               IF NOT "Valves_DB".Valve[#i].Healthy OR "Valves_DB".PositionFault[#i]
                  OR "Valves_DB".TimeoutOpenAlarm[#i] OR "Valves_DB".TimeoutCloseAlarm[#i]
                  OR "Valves_DB".UnexpMove[#i] OR "Valves_DB".PosLostTmr[#i].Q
                  OR "Valves_DB".DirFault[#i] THEN
                   "Valves_DB".StateCode[#i] := 1;
                   #tempFault := #tempFault + 1;
                   IF #i <= 27 THEN #tempAftFault := #tempAftFault + 1;
                   ELSIF #i <= 54 THEN #tempErFault := #tempErFault + 1;
                   ELSE #tempFwdFault := #tempFwdFault + 1;
                   END_IF;
               ELSIF "Valves_DB".Valve[#i].LocalMode THEN
                   "Valves_DB".StateCode[#i] := 2;
                   #tempLocal := #tempLocal + 1;
                   IF #i <= 27 THEN #tempAftLocal := #tempAftLocal + 1;
                   ELSIF #i <= 54 THEN #tempErLocal := #tempErLocal + 1;
                   ELSE #tempFwdLocal := #tempFwdLocal + 1;
                   END_IF;
               ELSIF "Valves_DB".Valve[#i].OpenValve THEN
                   // 6 = OPENING. The run latches are checked BEFORE the limit switches on purpose:
                   // what the system is doing to the valve outranks where the valve currently sits.
                   // Without this, a valve commanded CLOSE while still on its open limit displayed a
                   // settled green "FULLY OPEN" - no acknowledgement that the command had even
                   // registered on a normal stroke, and on a fault a confidently wrong indication for
                   // the full travel timeout. StateCode used to answer only "where is the valve";
                   // it now also answers "what is being done to it", which is the half that matters
                   // when something is going wrong.
                   "Valves_DB".StateCode[#i] := 6;
                   #tempTransit := #tempTransit + 1;
                   IF #i <= 27 THEN #tempAftTransit := #tempAftTransit + 1;
                   ELSIF #i <= 54 THEN #tempErTransit := #tempErTransit + 1;
                   ELSE #tempFwdTransit := #tempFwdTransit + 1;
                   END_IF;
               ELSIF "Valves_DB".Valve[#i].CloseValve THEN
                   "Valves_DB".StateCode[#i] := 7;   // 7 = CLOSING
                   #tempTransit := #tempTransit + 1;
                   IF #i <= 27 THEN #tempAftTransit := #tempAftTransit + 1;
                   ELSIF #i <= 54 THEN #tempErTransit := #tempErTransit + 1;
                   ELSE #tempFwdTransit := #tempFwdTransit + 1;
                   END_IF;
               ELSIF "Valves_DB".Valve[#i].OpenFB AND NOT "Valves_DB".Valve[#i].ClosedFB THEN
                   "Valves_DB".StateCode[#i] := 3;
                   #tempOpen := #tempOpen + 1;
                   IF #i <= 27 THEN #tempAftOpen := #tempAftOpen + 1;
                   ELSIF #i <= 54 THEN #tempErOpen := #tempErOpen + 1;
                   ELSE #tempFwdOpen := #tempFwdOpen + 1;
                   END_IF;
               ELSIF NOT "Valves_DB".Valve[#i].OpenFB AND "Valves_DB".Valve[#i].ClosedFB THEN
                   "Valves_DB".StateCode[#i] := 4;
                   #tempClosed := #tempClosed + 1;
                   IF #i <= 27 THEN #tempAftClosed := #tempAftClosed + 1;
                   ELSIF #i <= 54 THEN #tempErClosed := #tempErClosed + 1;
                   ELSE #tempFwdClosed := #tempFwdClosed + 1;
                   END_IF;
               ELSE
                   "Valves_DB".StateCode[#i] := 5;
                   #tempTransit := #tempTransit + 1; // MOVING state!
                   IF #i <= 27 THEN #tempAftTransit := #tempAftTransit + 1;
                   ELSIF #i <= 54 THEN #tempErTransit := #tempErTransit + 1;
                   ELSE #tempFwdTransit := #tempFwdTransit + 1;
                   END_IF;
               END_IF;
           ELSE
               "Valves_DB".StateCode[#i] := 0;
               "Valves_DB".PosCode[#i] := 0;
               "Valves_DB".DispCode[#i] := 0;
               "Valves_DB".FaultCode[#i] := 0;
               "Valves_DB".Valve[#i].OpenCmd := FALSE;
               "Valves_DB".Valve[#i].CloseCmd := FALSE;
               // Drop the run latches too. Without this, de-configuring a valve mid-travel (the popup's
               // SERVICE toggle reaches this from the HMI) left OpenValve/CloseValve latched TRUE with
               // no logic left managing them - and since FC_IoMapper skipped unconfigured valves, the
               // DQ bit kept its last value and FC_PhysicalIoCopy went on copying it to the real %Q
               // forever. The relay would have stayed energised indefinitely while the screen showed a
               // harmless-looking UNCONFIGURED. Paired with the FC_IoMapper change that now drives DQ
               // unconditionally, so clearing these actually de-energises the output.
               "Valves_DB".Valve[#i].OpenValve := FALSE;
               "Valves_DB".Valve[#i].CloseValve := FALSE;
               "Valves_DB".CmdPos[#i] := 0;
               // Don't let an unconfigured/removed valve leave a stale latched alarm behind.
               "Valves_DB".TimeoutOpenAlarm[#i] := FALSE;
               "Valves_DB".TimeoutCloseAlarm[#i] := FALSE;
               "Valves_DB".UnexpMove[#i] := FALSE;
               "Valves_DB".DirFault[#i] := FALSE;
               "Valves_DB".PrevOpenFB[#i] := FALSE;
               "Valves_DB".PrevClosedFB[#i] := FALSE;
           END_IF;
       END_FOR;

       "Valves_DB".TotalOpen := #tempOpen;
       "Valves_DB".TotalClosed := #tempClosed;
       "Valves_DB".TotalTransit := #tempTransit;
       "Valves_DB".TotalFault := #tempFault;
       "Valves_DB".TotalLocal := #tempLocal;
       "Valves_DB".TotalConfigured := #tempConfigured;

       "Valves_DB".ErOpen := #tempErOpen;
       "Valves_DB".ErClosed := #tempErClosed;
       "Valves_DB".ErTransit := #tempErTransit;
       "Valves_DB".ErFault := #tempErFault;
       "Valves_DB".ErLocal := #tempErLocal;
       "Valves_DB".ErConfigured := #tempErConfigured;

       "Valves_DB".FwdOpen := #tempFwdOpen;
       "Valves_DB".FwdClosed := #tempFwdClosed;
       "Valves_DB".FwdTransit := #tempFwdTransit;
       "Valves_DB".FwdFault := #tempFwdFault;
       "Valves_DB".FwdLocal := #tempFwdLocal;
       "Valves_DB".FwdConfigured := #tempFwdConfigured;

       "Valves_DB".AftOpen := #tempAftOpen;
       "Valves_DB".AftClosed := #tempAftClosed;
       "Valves_DB".AftTransit := #tempAftTransit;
       "Valves_DB".AftFault := #tempAftFault;
       "Valves_DB".AftLocal := #tempAftLocal;
       "Valves_DB".AftConfigured := #tempAftConfigured;

       // ---- Alarm condition bit-packing -----------------------------------------
       // WinCC discrete alarms trigger off a bit within a Word tag (RaisedStateTag +
       // RaisedStateTagBitNumber), not a bare Bool array element, so each of the 7 per-valve
       // conditions gets packed into 6 words (96 bits available, 89 used) here. Valve V's bit for any
       // condition is word (V-1)/16, bit (V-1) MOD 16 — matches how the HMI-side alarm creation
       // computes the same trigger address, so the two have to stay in lockstep.
       FOR #w := 0 TO 5 DO
           #packWord := 0;
           FOR #b := 0 TO 15 DO
               #bitIdx := #w * 16 + #b + 1;
               IF #bitIdx <= 89 THEN
                   IF "Valves_DB".Valve[#bitIdx].Configured AND NOT "Valves_DB".Valve[#bitIdx].Healthy THEN
                       #packWord := #packWord OR SHL(IN := W#16#1, N := INT_TO_UDINT(#b));
                   END_IF;
               END_IF;
           END_FOR;
           "Valves_DB".W_Unhealthy[#w] := #packWord;
       END_FOR;

       FOR #w := 0 TO 5 DO
           #packWord := 0;
           FOR #b := 0 TO 15 DO
               #bitIdx := #w * 16 + #b + 1;
               IF #bitIdx <= 89 THEN
                   IF "Valves_DB".Valve[#bitIdx].Configured AND "Valves_DB".Valve[#bitIdx].OpenFB AND "Valves_DB".Valve[#bitIdx].ClosedFB THEN
                       #packWord := #packWord OR SHL(IN := W#16#1, N := INT_TO_UDINT(#b));
                   END_IF;
               END_IF;
           END_FOR;
           "Valves_DB".W_Conflict[#w] := #packWord;
       END_FOR;

       FOR #w := 0 TO 5 DO
           #packWord := 0;
           FOR #b := 0 TO 15 DO
               #bitIdx := #w * 16 + #b + 1;
               IF #bitIdx <= 89 THEN
                   IF "Valves_DB".Valve[#bitIdx].Configured AND "Valves_DB".TimeoutOpenAlarm[#bitIdx] THEN
                       #packWord := #packWord OR SHL(IN := W#16#1, N := INT_TO_UDINT(#b));
                   END_IF;
               END_IF;
           END_FOR;
           "Valves_DB".W_FailOpen[#w] := #packWord;
       END_FOR;

       FOR #w := 0 TO 5 DO
           #packWord := 0;
           FOR #b := 0 TO 15 DO
               #bitIdx := #w * 16 + #b + 1;
               IF #bitIdx <= 89 THEN
                   IF "Valves_DB".Valve[#bitIdx].Configured AND "Valves_DB".TimeoutCloseAlarm[#bitIdx] THEN
                       #packWord := #packWord OR SHL(IN := W#16#1, N := INT_TO_UDINT(#b));
                   END_IF;
               END_IF;
           END_FOR;
           "Valves_DB".W_FailClose[#w] := #packWord;
       END_FOR;

       FOR #w := 0 TO 5 DO
           #packWord := 0;
           FOR #b := 0 TO 15 DO
               #bitIdx := #w * 16 + #b + 1;
               IF #bitIdx <= 89 THEN
                   IF "Valves_DB".Valve[#bitIdx].Configured AND "Valves_DB".PosLostTmr[#bitIdx].Q THEN
                       #packWord := #packWord OR SHL(IN := W#16#1, N := INT_TO_UDINT(#b));
                   END_IF;
               END_IF;
           END_FOR;
           "Valves_DB".W_LossPos[#w] := #packWord;
       END_FOR;

       FOR #w := 0 TO 5 DO
           #packWord := 0;
           FOR #b := 0 TO 15 DO
               #bitIdx := #w * 16 + #b + 1;
               IF #bitIdx <= 89 THEN
                   IF "Valves_DB".Valve[#bitIdx].Configured AND "Valves_DB".UnexpMove[#bitIdx] THEN
                       #packWord := #packWord OR SHL(IN := W#16#1, N := INT_TO_UDINT(#b));
                   END_IF;
               END_IF;
           END_FOR;
           "Valves_DB".W_UnexpMove[#w] := #packWord;
       END_FOR;

       FOR #w := 0 TO 5 DO
           #packWord := 0;
           FOR #b := 0 TO 15 DO
               #bitIdx := #w * 16 + #b + 1;
               IF #bitIdx <= 89 THEN
                   IF "Valves_DB".Valve[#bitIdx].Configured AND "Valves_DB".Valve[#bitIdx].LocalMode THEN
                       #packWord := #packWord OR SHL(IN := W#16#1, N := INT_TO_UDINT(#b));
                   END_IF;
               END_IF;
           END_FOR;
           "Valves_DB".W_Local[#w] := #packWord;
       END_FOR;

       // H: direction / limit-switch discrepancy.
       FOR #w := 0 TO 5 DO
           #packWord := 0;
           FOR #b := 0 TO 15 DO
               #bitIdx := #w * 16 + #b + 1;
               IF #bitIdx <= 89 THEN
                   IF "Valves_DB".Valve[#bitIdx].Configured AND "Valves_DB".DirFault[#bitIdx] THEN
                       #packWord := #packWord OR SHL(IN := W#16#1, N := INT_TO_UDINT(#b));
                   END_IF;
               END_IF;
           END_FOR;
           "Valves_DB".W_DirFault[#w] := #packWord;
       END_FOR;

       // Simulated hardware health (indices 1..9) into a single word.
       #packWord := 0;
       FOR #b := 0 TO 8 DO
           IF NOT "Valves_DB".HwHealthy[#b + 1] THEN
               #packWord := #packWord OR SHL(IN := W#16#1, N := INT_TO_UDINT(#b));
           END_IF;
       END_FOR;
       "Valves_DB".HwWord := #packWord;

       // ---- Paged table windows ------------------------------------------------
       // The HMI valve table has 14 fixed slots. Copy whichever page each zone is showing into
       // these windows so every HMI slot can bind to a constant tag name (e.g. ErTblState[3])
       // rather than building the name in JavaScript from a page tag — that indirection is what
       // forced the table onto ~126 polled scripts and made the screen slow to load.
       // TblState = -1 marks a slot with no valve on this page (0 already means UNCONFIGURED).
       // 14 iterations x 3 zones per scan is negligible next to the 89-valve loop above.

       // ── PAGED TABLE WINDOWS — gated, not rebuilt every scan ────────────────────────────
       // These four loops copy ~350 STRINGS per scan (tag, name, location, function, CmNo, VTag,
       // state text x 58 slots). String copies are the slowest thing in this program and were the
       // single biggest contributor to scan time, all to produce data no operator can read faster
       // than a few times a second.
       // So: rebuild on a 200 ms tick, OR immediately when a page changes. The page test matters -
       // waiting up to 200 ms after a page button would feel laggy, and paging is the one moment the
       // window contents change wholesale.
       #doWindows := #winTick
           OR ("Valves_DB".AftPage <> "Valves_DB".PrevAftPage)
           OR ("Valves_DB".ErPage  <> "Valves_DB".PrevErPage)
           OR ("Valves_DB".FwdPage <> "Valves_DB".PrevFwdPage)
           OR ("Valves_DB".CfgPage <> "Valves_DB".PrevCfgPage);

       IF #doWindows THEN
           "Valves_DB".PrevAftPage := "Valves_DB".AftPage;
           "Valves_DB".PrevErPage  := "Valves_DB".ErPage;
           "Valves_DB".PrevFwdPage := "Valves_DB".FwdPage;
           "Valves_DB".PrevCfgPage := "Valves_DB".CfgPage;

           // AFT BALLAST: valves 1..27 (2 pages)
           #base := 1 + "Valves_DB".AftPage * 14;
           FOR #j := 1 TO 14 DO
               #idx := #base + #j - 1;
               IF #idx <= 27 THEN
                   "Valves_DB".AftTblState[#j] := "Valves_DB".StateCode[#idx];
                   "Valves_DB".AftTblNo[#j] := #idx;
                   // RIGHT() strips the leading sign-space INT_TO_STRING puts in front of a positive
                   // number: without it CONCAT yields 'CM- 29' rather than 'CM-29'.
                   IF #idx < 10 THEN
                       "Valves_DB".AftTblTag[#j] := CONCAT(IN1 := 'CM-0', IN2 := RIGHT(IN := INT_TO_STRING(#idx), L := 1));
                   ELSE
                       "Valves_DB".AftTblTag[#j] := CONCAT(IN1 := 'CM-', IN2 := RIGHT(IN := INT_TO_STRING(#idx), L := 2));
                   END_IF;
                   "Valve_Meta_DB".AftTblName[#j] := "Valve_Meta_DB".Name[#idx];
                   "Valve_Meta_DB".AftTblLoc[#j] := "Valve_Meta_DB".Location[#idx];
                   "Valve_Meta_DB".AftTblFunc[#j] := "Valve_Meta_DB".FuncName[#idx];
                   "Valve_Meta_DB".AftTblCmNo[#j] := "Valve_Meta_DB".CmNo[#idx];
                   "Valve_Meta_DB".AftTblVTag[#j] := "Valve_Meta_DB".VTag[#idx];
                   CASE "Valves_DB".StateCode[#idx] OF
                       0: "Valves_DB".AftTblStateTxt[#j] := 'UNCONFIGURED';
                       1: "Valves_DB".AftTblStateTxt[#j] := 'FAULT';
                       2: "Valves_DB".AftTblStateTxt[#j] := 'LOCAL';
                       3: "Valves_DB".AftTblStateTxt[#j] := 'OPEN';
                       4: "Valves_DB".AftTblStateTxt[#j] := 'CLOSED';
                       6: "Valves_DB".AftTblStateTxt[#j] := 'OPENING';
                       7: "Valves_DB".AftTblStateTxt[#j] := 'CLOSING';
                       // 'NO POSITION', not 'MOVING'. Code 5 means neither limit switch is made, which is
                       // not the same as motion - 6 and 7 carry the genuine motion states now. Observed
                       // live 2026-08-16: after Reset Fault on a failed travel the valve sits perfectly
                       // still with no position for the 2s Loss-of-Position debounce, and the panel read
                       // MOVING. That is the one moment the operator most needs the truth.
                       ELSE "Valves_DB".AftTblStateTxt[#j] := 'NO POSITION';
                   END_CASE;
               ELSE
                   // 9, not 6: 6 became a real StateCode (OPENING) on 2026-08-16, and this
                   // empty-slot sentinel shares the same value map on the HMI. Leaving it at 6 painted
                   // every opening valve's status text transparent. 9 is outside the StateCode range.
                   "Valves_DB".AftTblState[#j] := 9;
                   "Valves_DB".AftTblNo[#j] := 0;
                   "Valves_DB".AftTblTag[#j] := '';
                   "Valves_DB".AftTblStateTxt[#j] := '';
                   "Valve_Meta_DB".AftTblName[#j] := '';
                   "Valve_Meta_DB".AftTblLoc[#j] := '';
                   "Valve_Meta_DB".AftTblFunc[#j] := '';
                   "Valve_Meta_DB".AftTblCmNo[#j] := '';
                   "Valve_Meta_DB".AftTblVTag[#j] := '';
               END_IF;
           END_FOR;

           // BILGE / ER: valves 28..54 (2 pages)
           #base := 28 + "Valves_DB".ErPage * 14;
           FOR #j := 1 TO 14 DO
               #idx := #base + #j - 1;
               IF #idx <= 54 THEN
                   "Valves_DB".ErTblState[#j] := "Valves_DB".StateCode[#idx];
                   "Valves_DB".ErTblNo[#j] := #idx - 27;
                   "Valves_DB".ErTblTag[#j] := CONCAT(IN1 := 'CM-', IN2 := RIGHT(IN := INT_TO_STRING(#idx), L := 2));
                   "Valve_Meta_DB".ErTblName[#j] := "Valve_Meta_DB".Name[#idx];
                   "Valve_Meta_DB".ErTblLoc[#j] := "Valve_Meta_DB".Location[#idx];
                   "Valve_Meta_DB".ErTblFunc[#j] := "Valve_Meta_DB".FuncName[#idx];
                   "Valve_Meta_DB".ErTblCmNo[#j] := "Valve_Meta_DB".CmNo[#idx];
                   "Valve_Meta_DB".ErTblVTag[#j] := "Valve_Meta_DB".VTag[#idx];
                   CASE "Valves_DB".StateCode[#idx] OF
                       0: "Valves_DB".ErTblStateTxt[#j] := 'UNCONFIGURED';
                       1: "Valves_DB".ErTblStateTxt[#j] := 'FAULT';
                       2: "Valves_DB".ErTblStateTxt[#j] := 'LOCAL';
                       3: "Valves_DB".ErTblStateTxt[#j] := 'OPEN';
                       4: "Valves_DB".ErTblStateTxt[#j] := 'CLOSED';
                       6: "Valves_DB".ErTblStateTxt[#j] := 'OPENING';
                       7: "Valves_DB".ErTblStateTxt[#j] := 'CLOSING';
                       ELSE "Valves_DB".ErTblStateTxt[#j] := 'NO POSITION';
                   END_CASE;
               ELSE
                   "Valves_DB".ErTblState[#j] := 9;   // empty slot — see AftTblState note above
                   "Valves_DB".ErTblNo[#j] := 0;
                   "Valves_DB".ErTblTag[#j] := '';
                   "Valves_DB".ErTblStateTxt[#j] := '';
                   "Valve_Meta_DB".ErTblName[#j] := '';
                   "Valve_Meta_DB".ErTblLoc[#j] := '';
                   "Valve_Meta_DB".ErTblFunc[#j] := '';
                   "Valve_Meta_DB".ErTblCmNo[#j] := '';
                   "Valve_Meta_DB".ErTblVTag[#j] := '';
               END_IF;
           END_FOR;

           // FORWARD BALLAST: valves 55..89 (3 pages of 14, 35 slots exactly - the widest zone, holding
           // the schedule's 35 FWD valves with no spare)
           #base := 55 + "Valves_DB".FwdPage * 14;
           FOR #j := 1 TO 14 DO
               #idx := #base + #j - 1;
               IF #idx <= 89 THEN
                   "Valves_DB".FwdTblState[#j] := "Valves_DB".StateCode[#idx];
                   "Valves_DB".FwdTblNo[#j] := #idx - 54;
                   "Valves_DB".FwdTblTag[#j] := CONCAT(IN1 := 'CM-', IN2 := RIGHT(IN := INT_TO_STRING(#idx), L := 2));
                   "Valve_Meta_DB".FwdTblName[#j] := "Valve_Meta_DB".Name[#idx];
                   "Valve_Meta_DB".FwdTblLoc[#j] := "Valve_Meta_DB".Location[#idx];
                   "Valve_Meta_DB".FwdTblFunc[#j] := "Valve_Meta_DB".FuncName[#idx];
                   "Valve_Meta_DB".FwdTblCmNo[#j] := "Valve_Meta_DB".CmNo[#idx];
                   "Valve_Meta_DB".FwdTblVTag[#j] := "Valve_Meta_DB".VTag[#idx];
                   CASE "Valves_DB".StateCode[#idx] OF
                       0: "Valves_DB".FwdTblStateTxt[#j] := 'UNCONFIGURED';
                       1: "Valves_DB".FwdTblStateTxt[#j] := 'FAULT';
                       2: "Valves_DB".FwdTblStateTxt[#j] := 'LOCAL';
                       3: "Valves_DB".FwdTblStateTxt[#j] := 'OPEN';
                       4: "Valves_DB".FwdTblStateTxt[#j] := 'CLOSED';
                       6: "Valves_DB".FwdTblStateTxt[#j] := 'OPENING';
                       7: "Valves_DB".FwdTblStateTxt[#j] := 'CLOSING';
                       ELSE "Valves_DB".FwdTblStateTxt[#j] := 'NO POSITION';
                   END_CASE;
               ELSE
                   "Valves_DB".FwdTblState[#j] := 9;   // empty slot — see AftTblState note above
                   "Valves_DB".FwdTblNo[#j] := 0;
                   "Valves_DB".FwdTblTag[#j] := '';
                   "Valves_DB".FwdTblStateTxt[#j] := '';
                   "Valve_Meta_DB".FwdTblName[#j] := '';
                   "Valve_Meta_DB".FwdTblLoc[#j] := '';
                   "Valve_Meta_DB".FwdTblFunc[#j] := '';
                   "Valve_Meta_DB".FwdTblCmNo[#j] := '';
                   "Valve_Meta_DB".FwdTblVTag[#j] := '';
               END_IF;
           END_FOR;

           // CONFIGURATION SCREEN: all 89 slots in one global sequence (6 pages of 16, last one ragged
           // at 9), not zone-scoped like the three windows above - this screen shows the whole fleet,
           // so #idx IS the absolute valve number directly, no zone-start offset needed.
           #base := 1 + "Valves_DB".CfgPage * 16;
           FOR #j := 1 TO 16 DO
               #idx := #base + #j - 1;
               IF #idx <= 89 THEN
                   "Valves_DB".CfgTblNo[#j] := #idx;
                   IF #idx < 10 THEN
                       "Valves_DB".CfgTblTag[#j] := CONCAT(IN1 := 'CM-0', IN2 := RIGHT(IN := INT_TO_STRING(#idx), L := 1));
                   ELSE
                       "Valves_DB".CfgTblTag[#j] := CONCAT(IN1 := 'CM-', IN2 := RIGHT(IN := INT_TO_STRING(#idx), L := 2));
                   END_IF;
                   IF #idx <= 27 THEN
                       "Valves_DB".CfgTblZone[#j] := 'AFT BALLAST';
                   ELSIF #idx <= 54 THEN
                       "Valves_DB".CfgTblZone[#j] := 'BILGE-ER';
                   ELSE
                       "Valves_DB".CfgTblZone[#j] := 'BALLAST FWD';
                   END_IF;
                   "Valve_Meta_DB".CfgTblName[#j] := "Valve_Meta_DB".Name[#idx];
                   "Valve_Meta_DB".CfgTblLoc[#j] := "Valve_Meta_DB".Location[#idx];
                   // Client-schedule identity columns. Displayed verbatim - no fallback to the
                   // computed CmNo/zone strings above, because a blank here is meaningful: it means
                   // that valve has not been entered from the confirmed schedule yet, and showing a
                   // derived 'CM-07' in its place would misrepresent unentered data as real.
                   "Valve_Meta_DB".CfgTblCmNo[#j] := "Valve_Meta_DB".CmNo[#idx];
                   "Valve_Meta_DB".CfgTblVTag[#j] := "Valve_Meta_DB".VTag[#idx];
                   "Valve_Meta_DB".CfgTblSys[#j] := "Valve_Meta_DB".SysName[#idx];
                   "Valve_Meta_DB".CfgTblFunc[#j] := "Valve_Meta_DB".FuncName[#idx];
                   "Valves_DB".CfgTblConfigured[#j] := "Valves_DB".Valve[#idx].Configured;
                   "Valves_DB".CfgTblState[#j] := "Valves_DB".StateCode[#idx];
                   CASE "Valves_DB".StateCode[#idx] OF
                       0: "Valves_DB".CfgTblStateTxt[#j] := 'UNCONFIGURED';
                       1: "Valves_DB".CfgTblStateTxt[#j] := 'FAULT';
                       2: "Valves_DB".CfgTblStateTxt[#j] := 'LOCAL';
                       3: "Valves_DB".CfgTblStateTxt[#j] := 'OPEN';
                       4: "Valves_DB".CfgTblStateTxt[#j] := 'CLOSED';
                       6: "Valves_DB".CfgTblStateTxt[#j] := 'OPENING';
                       7: "Valves_DB".CfgTblStateTxt[#j] := 'CLOSING';
                       ELSE "Valves_DB".CfgTblStateTxt[#j] := 'NO POSITION';
                   END_CASE;
               ELSE
                   "Valves_DB".CfgTblNo[#j] := 0;
                   "Valves_DB".CfgTblTag[#j] := '';
                   "Valves_DB".CfgTblZone[#j] := '';
                   "Valve_Meta_DB".CfgTblName[#j] := '';
                   "Valve_Meta_DB".CfgTblLoc[#j] := '';
                   "Valve_Meta_DB".CfgTblCmNo[#j] := '';
                   "Valve_Meta_DB".CfgTblVTag[#j] := '';
                   "Valve_Meta_DB".CfgTblSys[#j] := '';
                   "Valve_Meta_DB".CfgTblFunc[#j] := '';
                   "Valves_DB".CfgTblConfigured[#j] := FALSE;
                   "Valves_DB".CfgTblState[#j] := 9;   // empty slot — see AftTblState note above
                   "Valves_DB".CfgTblStateTxt[#j] := '';
               END_IF;
           END_FOR;
       END_IF;


       // SELECTED-VALVE MIRROR for the control popup - same trick as the three paged table windows
       // above, applied to a window of exactly one valve. The HMI writes SelIdx when a valve badge is
       // tapped; this copies that valve's live fields into fixed, non-indexed tags.
       //
       // Why: every popup field used to compute its own tag name at runtime ("V" + idx + "_State"),
       // which WinCC cannot bind natively - so each one ran as a polled JavaScript at T500ms, ~14 of
       // them, and the popup visibly lagged on open and on switching valves. Reading fixed tag names
       // lets those same scripts run on AutomaticTags instead: evaluated when a value actually
       // changes, not on a timer. Zero polling, instant update.
       //
       // Out-of-range (including SelIdx = 0 before any valve has ever been tapped) yields the
       // unconfigured/blank state rather than stale data from whatever was selected last.
       #sel := "Valves_DB".SelIdx;
       IF #sel >= 1 AND #sel <= 89 THEN
           "Valves_DB".SelState      := "Valves_DB".StateCode[#sel];
           "Valves_DB".SelHealthy    := "Valves_DB".Valve[#sel].Healthy;
           "Valves_DB".SelLocalMode  := "Valves_DB".Valve[#sel].LocalMode;
           "Valves_DB".SelConfigured := "Valves_DB".Valve[#sel].Configured;
           "Valves_DB".SelDirFault   := "Valves_DB".DirFault[#sel];
           "Valves_DB".SelPositionFault := "Valves_DB".PositionFault[#sel];
           "Valves_DB".SelCmdPos     := "Valves_DB".CmdPos[#sel];
           "Valves_DB".SelPosCode    := "Valves_DB".PosCode[#sel];
           "Valves_DB".SelFaultCode  := "Valves_DB".FaultCode[#sel];
           "Valve_Meta_DB".SelCmNo   := "Valve_Meta_DB".CmNo[#sel];
           "Valve_Meta_DB".SelVTag   := "Valve_Meta_DB".VTag[#sel];
       ELSE
           "Valves_DB".SelState      := 0;
           "Valves_DB".SelHealthy    := FALSE;
           "Valves_DB".SelLocalMode  := FALSE;
           "Valves_DB".SelConfigured := FALSE;
           "Valves_DB".SelDirFault   := FALSE;
           "Valves_DB".SelPositionFault := FALSE;
           "Valves_DB".SelCmdPos     := 0;
           "Valves_DB".SelPosCode    := 0;
           "Valves_DB".SelFaultCode  := 0;
           "Valve_Meta_DB".SelCmNo   := '';
           "Valve_Meta_DB".SelVTag   := '';
       END_IF;
END_FUNCTION_BLOCK

FUNCTION "FC_PhysicalIoCopy" : Void   // FC2, SCL
{ S7_Optimized_Access := 'TRUE' }
VERSION : 0.1
// NOT YET WIRED INTO Main[OB1]. Generated 2026-08-08 from the real addresses confirmed live in TIA's Device overview after assigning all 3 ET200SP stations (AFT/MID/FWD) to PLC_1's PROFINET IO system - before that, every module showed no address at all. This is the only block in the whole project that references real physical %I/%Q addresses; everything downstream (FC_IoMapper, Valve_Channels_DB) only ever deals with the abstract 1..368 / 1..208 channel numbers in IO_Buffer_DB. Still needs: (1) FB_ValveLoop simulation guard for real-mapped valves, (2) both this and FC_IoMapper actually called from Main[OB1] - see FC_IoMapper's own header comment. Safe to have present unwired: it only touches IO_Buffer_DB, which nothing else reads yet.
// stored: AutoNumber true, IsIECCheckEnabled false, SetENOAutomatically false, UDAEnableTagReadback false
BEGIN
// Network 1

       // === DIGITAL INPUTS: real %I bits -> IO_Buffer_DB.DI[1..368] ===
       // -- AFT DI modules --
       "IO_Buffer_DB".DI[1] := "Tag__639217692550262421";
       "IO_Buffer_DB".DI[2] := "Tag__639217692553776870";
       "IO_Buffer_DB".DI[3] := "Tag__639217692553954872";
       "IO_Buffer_DB".DI[4] := "Tag__639217692553954873";
       "IO_Buffer_DB".DI[5] := "Tag__639217692554216438";
       "IO_Buffer_DB".DI[6] := "Tag__639217692554394622";
       "IO_Buffer_DB".DI[7] := "Tag__639217692554432300";
       "IO_Buffer_DB".DI[8] := "Tag__639217692556336031";
       "IO_Buffer_DB".DI[9] := "Tag__639217692556550149";
       "IO_Buffer_DB".DI[10] := "Tag__639217692556680608";
       "IO_Buffer_DB".DI[11] := "Tag__639217692556821735";
       "IO_Buffer_DB".DI[12] := "Tag__639217692556891742";
       "IO_Buffer_DB".DI[13] := "Tag__639217692557049682";
       "IO_Buffer_DB".DI[14] := "Tag__639217692557209508";
       "IO_Buffer_DB".DI[15] := "Tag__639217692557209509";
       "IO_Buffer_DB".DI[16] := "Tag__639217692557471753";
       "IO_Buffer_DB".DI[17] := "Tag__639217692557529414";
       "IO_Buffer_DB".DI[18] := "Tag__639217692557689863";
       "IO_Buffer_DB".DI[19] := "Tag__639217692557850060";
       "IO_Buffer_DB".DI[20] := "Tag__639217692558010331";
       "IO_Buffer_DB".DI[21] := "Tag__639217692558171799";
       "IO_Buffer_DB".DI[22] := "Tag__639217692558331401";
       "IO_Buffer_DB".DI[23] := "Tag__639217692558488410";
       "IO_Buffer_DB".DI[24] := "Tag__639217692558802162";
       "IO_Buffer_DB".DI[25] := "Tag__639217692558961456";
       "IO_Buffer_DB".DI[26] := "Tag__639217692558971616";
       "IO_Buffer_DB".DI[27] := "Tag__639217692559129482";
       "IO_Buffer_DB".DI[28] := "Tag__639217692559281543";
       "IO_Buffer_DB".DI[29] := "Tag__639217692559443162";
       "IO_Buffer_DB".DI[30] := "Tag__639217692559601745";
       "IO_Buffer_DB".DI[31] := "Tag__639217692559760896";
       "IO_Buffer_DB".DI[32] := "Tag__639217692559921432";
       "IO_Buffer_DB".DI[33] := "Tag__639217692559921433";
       "IO_Buffer_DB".DI[34] := "Tag__639217692560082018";
       "IO_Buffer_DB".DI[35] := "Tag__639217692560402934";
       "IO_Buffer_DB".DI[36] := "Tag__639217692560402935";
       "IO_Buffer_DB".DI[37] := "Tag__639217692560583987";
       "IO_Buffer_DB".DI[38] := "Tag__639217692560723706";
       "IO_Buffer_DB".DI[39] := "Tag__639217692560880740";
       "IO_Buffer_DB".DI[40] := "Tag__639217692561041807";
       "IO_Buffer_DB".DI[41] := "Tag__639217692561206457";
       "IO_Buffer_DB".DI[42] := "Tag__639217692561359218";
       "IO_Buffer_DB".DI[43] := "Tag__639217692561520184";
       "IO_Buffer_DB".DI[44] := "Tag__639217692561520185";
       "IO_Buffer_DB".DI[45] := "Tag__639217692561802187";
       "IO_Buffer_DB".DI[46] := "Tag__639217692561935087";
       "IO_Buffer_DB".DI[47] := "Tag__639217692562065024";
       "IO_Buffer_DB".DI[48] := "Tag__639217692562223286";
       "IO_Buffer_DB".DI[49] := "Tag__639217692562383723";
       "IO_Buffer_DB".DI[50] := "Tag__639217692562543936";
       "IO_Buffer_DB".DI[51] := "Tag__639217692562543937";
       "IO_Buffer_DB".DI[52] := "Tag__639217692562862407";
       "IO_Buffer_DB".DI[53] := "Tag__639217692562862408";
       "IO_Buffer_DB".DI[54] := "Tag__639217692563093001";
       "IO_Buffer_DB".DI[55] := "Tag__639217692563182212";
       "IO_Buffer_DB".DI[56] := "Tag__639217692563343596";
       "IO_Buffer_DB".DI[57] := "Tag__639217692563511187";
       "IO_Buffer_DB".DI[58] := "Tag__639217692563662093";
       "IO_Buffer_DB".DI[59] := "Tag__639217692563662094";
       "IO_Buffer_DB".DI[60] := "Tag__639217692563823907";
       "IO_Buffer_DB".DI[61] := "Tag__639217692566083593";
       "IO_Buffer_DB".DI[62] := "Tag__639217692566201557";
       "IO_Buffer_DB".DI[63] := "Tag__639217692566360040";
       "IO_Buffer_DB".DI[64] := "Tag__639217692566517145";
       "IO_Buffer_DB".DI[65] := "Tag__639217692566674032";
       "IO_Buffer_DB".DI[66] := "Tag__639217692566832496";
       "IO_Buffer_DB".DI[67] := "Tag__639217692566832497";
       "IO_Buffer_DB".DI[68] := "Tag__639217692567184922";
       "IO_Buffer_DB".DI[69] := "Tag__639217692567336780";
       "IO_Buffer_DB".DI[70] := "Tag__639217692567388945";
       "IO_Buffer_DB".DI[71] := "Tag__639217692567546587";
       "IO_Buffer_DB".DI[72] := "Tag__639217692567707146";
       "IO_Buffer_DB".DI[73] := "Tag__639217692567868007";
       "IO_Buffer_DB".DI[74] := "Tag__639217692567868008";
       "IO_Buffer_DB".DI[75] := "Tag__639217692568025035";
       "IO_Buffer_DB".DI[76] := "Tag__639217692568182907";
       "IO_Buffer_DB".DI[77] := "Tag__639217692568341074";
       "IO_Buffer_DB".DI[78] := "Tag__639217692568550097";
       "IO_Buffer_DB".DI[79] := "Tag__639217692568683019";
       "IO_Buffer_DB".DI[80] := "Tag__639217692568840948";
       "IO_Buffer_DB".DI[81] := "Tag__639217692568971320";
       "IO_Buffer_DB".DI[82] := "Tag__639217692569119475";
       "IO_Buffer_DB".DI[83] := "Tag__639217692569298523";
       "IO_Buffer_DB".DI[84] := "Tag__639217692569460008";
       "IO_Buffer_DB".DI[85] := "Tag__639217692569619373";
       "IO_Buffer_DB".DI[86] := "Tag__639217692569780777";
       "IO_Buffer_DB".DI[87] := "Tag__639217692569780778";
       "IO_Buffer_DB".DI[88] := "Tag__639217692569942097";
       "IO_Buffer_DB".DI[89] := "Tag__639217692570102018";
       "IO_Buffer_DB".DI[90] := "Tag__639217692570262026";
       "IO_Buffer_DB".DI[91] := "Tag__639217692570422186";
       "IO_Buffer_DB".DI[92] := "Tag__639217692570422187";
       "IO_Buffer_DB".DI[93] := "Tag__639217692570583489";
       "IO_Buffer_DB".DI[94] := "Tag__639217692570745102";
       "IO_Buffer_DB".DI[95] := "Tag__639217692570906074";
       "IO_Buffer_DB".DI[96] := "Tag__639217692570906075";
       "IO_Buffer_DB".DI[97] := "Tag__639217692571063660";
       "IO_Buffer_DB".DI[98] := "Tag__639217692571223097";
       "IO_Buffer_DB".DI[99] := "Tag__639217692571384739";
       "IO_Buffer_DB".DI[100] := "Tag__639217692571544096";
       "IO_Buffer_DB".DI[101] := "Tag__639217692571703825";
       "IO_Buffer_DB".DI[102] := "Tag__639217692571865026";
       "IO_Buffer_DB".DI[103] := "Tag__639217692572024808";
       "IO_Buffer_DB".DI[104] := "Tag__639217692572184903";
       "IO_Buffer_DB".DI[105] := "Tag__639217692572395679";
       "IO_Buffer_DB".DI[106] := "Tag__639217692572536054";
       "IO_Buffer_DB".DI[107] := "Tag__639217692572670856";
       "IO_Buffer_DB".DI[108] := "Tag__639217692572707880";
       "IO_Buffer_DB".DI[109] := "Tag__639217692572861963";
       "IO_Buffer_DB".DI[110] := "Tag__639217692573067363";
       "IO_Buffer_DB".DI[111] := "Tag__639217692573180541";
       "IO_Buffer_DB".DI[112] := "Tag__639217692573357884";
       // -- MID DI modules --
       "IO_Buffer_DB".DI[113] := "Tag__639217692573503474";
       "IO_Buffer_DB".DI[114] := "Tag__639217692573503475";
       "IO_Buffer_DB".DI[115] := "Tag__639217692573691090";
       "IO_Buffer_DB".DI[116] := "Tag__639217692573812370";
       "IO_Buffer_DB".DI[117] := "Tag__639217692573973083";
       "IO_Buffer_DB".DI[118] := "Tag__639217692574133186";
       "IO_Buffer_DB".DI[119] := "Tag__639217692574289638";
       "IO_Buffer_DB".DI[120] := "Tag__639217692574448526";
       "IO_Buffer_DB".DI[121] := "Tag__639217692574609334";
       "IO_Buffer_DB".DI[122] := "Tag__639217692574768434";
       "IO_Buffer_DB".DI[123] := "Tag__639217692574930294";
       "IO_Buffer_DB".DI[124] := "Tag__639217692575083184";
       "IO_Buffer_DB".DI[125] := "Tag__639217692575261129";
       "IO_Buffer_DB".DI[126] := "Tag__639217692575419042";
       "IO_Buffer_DB".DI[127] := "Tag__639217692575539382";
       "IO_Buffer_DB".DI[128] := "Tag__639217692575911602";
       "IO_Buffer_DB".DI[129] := "Tag__639217692576029509";
       "IO_Buffer_DB".DI[130] := "Tag__639217692576029510";
       "IO_Buffer_DB".DI[131] := "Tag__639217692576190207";
       "IO_Buffer_DB".DI[132] := "Tag__639217692576351259";
       "IO_Buffer_DB".DI[133] := "Tag__639217692576511022";
       "IO_Buffer_DB".DI[134] := "Tag__639217692576672087";
       "IO_Buffer_DB".DI[135] := "Tag__639217692576832345";
       "IO_Buffer_DB".DI[136] := "Tag__639217692576952866";
       "IO_Buffer_DB".DI[137] := "Tag__639217692576990475";
       "IO_Buffer_DB".DI[138] := "Tag__639217692577151896";
       "IO_Buffer_DB".DI[139] := "Tag__639217692577372028";
       "IO_Buffer_DB".DI[140] := "Tag__639217692577469814";
       "IO_Buffer_DB".DI[141] := "Tag__639217692577766896";
       "IO_Buffer_DB".DI[142] := "Tag__639217692577926746";
       "IO_Buffer_DB".DI[143] := "Tag__639217692578046402";
       "IO_Buffer_DB".DI[144] := "Tag__639217692578046403";
       "IO_Buffer_DB".DI[145] := "Tag__639217692578204423";
       "IO_Buffer_DB".DI[146] := "Tag__639217692578364346";
       "IO_Buffer_DB".DI[147] := "Tag__639217692578525327";
       "IO_Buffer_DB".DI[148] := "Tag__639217692578706091";
       "IO_Buffer_DB".DI[149] := "Tag__639217692578841403";
       "IO_Buffer_DB".DI[150] := "Tag__639217692579004858";
       "IO_Buffer_DB".DI[151] := "Tag__639217692579155731";
       "IO_Buffer_DB".DI[152] := "Tag__639217692579314254";
       "IO_Buffer_DB".DI[153] := "Tag__639217692579314255";
       "IO_Buffer_DB".DI[154] := "Tag__639217692579474584";
       "IO_Buffer_DB".DI[155] := "Tag__639217692579635203";
       "IO_Buffer_DB".DI[156] := "Tag__639217692579794995";
       "IO_Buffer_DB".DI[157] := "Tag__639217692579955090";
       "IO_Buffer_DB".DI[158] := "Tag__639217692580275677";
       "IO_Buffer_DB".DI[159] := "Tag__639217692580432274";
       "IO_Buffer_DB".DI[160] := "Tag__639217692580552766";
       "IO_Buffer_DB".DI[161] := "Tag__639217692580590363";
       "IO_Buffer_DB".DI[162] := "Tag__639217692580751532";
       "IO_Buffer_DB".DI[163] := "Tag__639217692580913166";
       "IO_Buffer_DB".DI[164] := "Tag__639217692581133835";
       "IO_Buffer_DB".DI[165] := "Tag__639217692581227406";
       "IO_Buffer_DB".DI[166] := "Tag__639217692581387294";
       "IO_Buffer_DB".DI[167] := "Tag__639217692581507780";
       "IO_Buffer_DB".DI[168] := "Tag__639217692581545371";
       "IO_Buffer_DB".DI[169] := "Tag__639217692581704532";
       "IO_Buffer_DB".DI[170] := "Tag__639217692581863905";
       "IO_Buffer_DB".DI[171] := "Tag__639217692581863906";
       "IO_Buffer_DB".DI[172] := "Tag__639217692582023588";
       "IO_Buffer_DB".DI[173] := "Tag__639217692582184822";
       "IO_Buffer_DB".DI[174] := "Tag__639217692582344335";
       "IO_Buffer_DB".DI[175] := "Tag__639217692582505209";
       "IO_Buffer_DB".DI[176] := "Tag__639217692582505210";
       "IO_Buffer_DB".DI[177] := "Tag__639217692582664098";
       "IO_Buffer_DB".DI[178] := "Tag__639217692582825326";
       "IO_Buffer_DB".DI[179] := "Tag__639217692582994863";
       "IO_Buffer_DB".DI[180] := "Tag__639217692583198482";
       "IO_Buffer_DB".DI[181] := "Tag__639217692583329182";
       "IO_Buffer_DB".DI[182] := "Tag__639217692583430354";
       "IO_Buffer_DB".DI[183] := "Tag__639217692583542618";
       "IO_Buffer_DB".DI[184] := "Tag__639217692583692939";
       "IO_Buffer_DB".DI[185] := "Tag__639217692585720764";
       "IO_Buffer_DB".DI[186] := "Tag__639217692585760931";
       "IO_Buffer_DB".DI[187] := "Tag__639217692585920591";
       "IO_Buffer_DB".DI[188] := "Tag__639217692586101165";
       "IO_Buffer_DB".DI[189] := "Tag__639217692586241395";
       "IO_Buffer_DB".DI[190] := "Tag__639217692586241396";
       "IO_Buffer_DB".DI[191] := "Tag__639217692586401865";
       "IO_Buffer_DB".DI[192] := "Tag__639217692586559348";
       "IO_Buffer_DB".DI[193] := "Tag__639217692586717642";
       "IO_Buffer_DB".DI[194] := "Tag__639217692586876705";
       "IO_Buffer_DB".DI[195] := "Tag__639217692587037050";
       "IO_Buffer_DB".DI[196] := "Tag__639217692587198156";
       "IO_Buffer_DB".DI[197] := "Tag__639217692587198157";
       "IO_Buffer_DB".DI[198] := "Tag__639217692587438593";
       "IO_Buffer_DB".DI[199] := "Tag__639217692587516326";
       "IO_Buffer_DB".DI[200] := "Tag__639217692587676973";
       "IO_Buffer_DB".DI[201] := "Tag__639217692587676974";
       "IO_Buffer_DB".DI[202] := "Tag__639217692587854158";
       "IO_Buffer_DB".DI[203] := "Tag__639217692587995295";
       "IO_Buffer_DB".DI[204] := "Tag__639217692588156000";
       "IO_Buffer_DB".DI[205] := "Tag__639217692588379878";
       "IO_Buffer_DB".DI[206] := "Tag__639217692588550268";
       "IO_Buffer_DB".DI[207] := "Tag__639217692588708101";
       "IO_Buffer_DB".DI[208] := "Tag__639217692588866833";
       "IO_Buffer_DB".DI[209] := "Tag__639217692589023179";
       "IO_Buffer_DB".DI[210] := "Tag__639217692589158483";
       "IO_Buffer_DB".DI[211] := "Tag__639217692589208458";
       "IO_Buffer_DB".DI[212] := "Tag__639217692589366891";
       "IO_Buffer_DB".DI[213] := "Tag__639217692589526977";
       "IO_Buffer_DB".DI[214] := "Tag__639217692589687241";
       "IO_Buffer_DB".DI[215] := "Tag__639217692589848658";
       "IO_Buffer_DB".DI[216] := "Tag__639217692589848659";
       "IO_Buffer_DB".DI[217] := "Tag__639217692590010039";
       "IO_Buffer_DB".DI[218] := "Tag__639217692590170658";
       "IO_Buffer_DB".DI[219] := "Tag__639217692590328833";
       "IO_Buffer_DB".DI[220] := "Tag__639217692590485955";
       "IO_Buffer_DB".DI[221] := "Tag__639217692590485956";
       "IO_Buffer_DB".DI[222] := "Tag__639217692590645258";
       "IO_Buffer_DB".DI[223] := "Tag__639217692590805752";
       "IO_Buffer_DB".DI[224] := "Tag__639217692590966425";
       // -- FWD DI modules --
       "IO_Buffer_DB".DI[225] := "Tag__639217692590966426";
       "IO_Buffer_DB".DI[226] := "Tag__639217692591127321";
       "IO_Buffer_DB".DI[227] := "Tag__639217692591285391";
       "IO_Buffer_DB".DI[228] := "Tag__639217692591446446";
       "IO_Buffer_DB".DI[229] := "Tag__639217692591605376";
       "IO_Buffer_DB".DI[230] := "Tag__639217692591923527";
       "IO_Buffer_DB".DI[231] := "Tag__639217692591923528";
       "IO_Buffer_DB".DI[232] := "Tag__639217692592084854";
       "IO_Buffer_DB".DI[233] := "Tag__639217692592246014";
       "IO_Buffer_DB".DI[234] := "Tag__639217692592406057";
       "IO_Buffer_DB".DI[235] := "Tag__639217692592406058";
       "IO_Buffer_DB".DI[236] := "Tag__639217692592567050";
       "IO_Buffer_DB".DI[237] := "Tag__639217692592727547";
       "IO_Buffer_DB".DI[238] := "Tag__639217692592888082";
       "IO_Buffer_DB".DI[239] := "Tag__639217692593114463";
       "IO_Buffer_DB".DI[240] := "Tag__639217692593206619";
       "IO_Buffer_DB".DI[241] := "Tag__639217692593364125";
       "IO_Buffer_DB".DI[242] := "Tag__639217692593535630";
       "IO_Buffer_DB".DI[243] := "Tag__639217692593656106";
       "IO_Buffer_DB".DI[244] := "Tag__639217692593702147";
       "IO_Buffer_DB".DI[245] := "Tag__639217692593935520";
       "IO_Buffer_DB".DI[246] := "Tag__639217692594074769";
       "IO_Buffer_DB".DI[247] := "Tag__639217692594204786";
       "IO_Buffer_DB".DI[248] := "Tag__639217692594204787";
       "IO_Buffer_DB".DI[249] := "Tag__639217692594365259";
       "IO_Buffer_DB".DI[250] := "Tag__639217692594522265";
       "IO_Buffer_DB".DI[251] := "Tag__639217692594681744";
       "IO_Buffer_DB".DI[252] := "Tag__639217692594681745";
       "IO_Buffer_DB".DI[253] := "Tag__639217692594842324";
       "IO_Buffer_DB".DI[254] := "Tag__639217692595003601";
       "IO_Buffer_DB".DI[255] := "Tag__639217692595162932";
       "IO_Buffer_DB".DI[256] := "Tag__639217692595295217";
       "IO_Buffer_DB".DI[257] := "Tag__639217692595321829";
       "IO_Buffer_DB".DI[258] := "Tag__639217692595479808";
       "IO_Buffer_DB".DI[259] := "Tag__639217692595637197";
       "IO_Buffer_DB".DI[260] := "Tag__639217692595797438";
       "IO_Buffer_DB".DI[261] := "Tag__639217692595959028";
       "IO_Buffer_DB".DI[262] := "Tag__639217692596136048";
       "IO_Buffer_DB".DI[263] := "Tag__639217692596337735";
       "IO_Buffer_DB".DI[264] := "Tag__639217692596435546";
       "IO_Buffer_DB".DI[265] := "Tag__639217692596435547";
       "IO_Buffer_DB".DI[266] := "Tag__639217692596596639";
       "IO_Buffer_DB".DI[267] := "Tag__639217692596754611";
       "IO_Buffer_DB".DI[268] := "Tag__639217692596914545";
       "IO_Buffer_DB".DI[269] := "Tag__639217692597075234";
       "IO_Buffer_DB".DI[270] := "Tag__639217692597075235";
       "IO_Buffer_DB".DI[271] := "Tag__639217692597235934";
       "IO_Buffer_DB".DI[272] := "Tag__639217692597397011";
       "IO_Buffer_DB".DI[273] := "Tag__639217692597554180";
       "IO_Buffer_DB".DI[274] := "Tag__639217692597711217";
       "IO_Buffer_DB".DI[275] := "Tag__639217692597871107";
       "IO_Buffer_DB".DI[276] := "Tag__639217692598028494";
       "IO_Buffer_DB".DI[277] := "Tag__639217692598185471";
       "IO_Buffer_DB".DI[278] := "Tag__639217692598185472";
       "IO_Buffer_DB".DI[279] := "Tag__639217692598345589";
       "IO_Buffer_DB".DI[280] := "Tag__639217692598572817";
       "IO_Buffer_DB".DI[281] := "Tag__639217692598703247";
       "IO_Buffer_DB".DI[282] := "Tag__639217692598865809";
       "IO_Buffer_DB".DI[283] := "Tag__639217692599003448";
       "IO_Buffer_DB".DI[284] := "Tag__639217692599080153";
       "IO_Buffer_DB".DI[285] := "Tag__639217692599295021";
       "IO_Buffer_DB".DI[286] := "Tag__639217692599434105";
       "IO_Buffer_DB".DI[287] := "Tag__639217692599574585";
       "IO_Buffer_DB".DI[288] := "Tag__639217692599692113";
       "IO_Buffer_DB".DI[289] := "Tag__639217692599852177";
       "IO_Buffer_DB".DI[290] := "Tag__639217692599852178";
       "IO_Buffer_DB".DI[291] := "Tag__639217692600013096";
       "IO_Buffer_DB".DI[292] := "Tag__639217692600225652";
       "IO_Buffer_DB".DI[293] := "Tag__639217692600329437";
       "IO_Buffer_DB".DI[294] := "Tag__639217692600517312";
       "IO_Buffer_DB".DI[295] := "Tag__639217692600648060";
       "IO_Buffer_DB".DI[296] := "Tag__639217692600809555";
       "IO_Buffer_DB".DI[297] := "Tag__639217692600970188";
       "IO_Buffer_DB".DI[298] := "Tag__639217692600970189";
       "IO_Buffer_DB".DI[299] := "Tag__639217692601290117";
       "IO_Buffer_DB".DI[300] := "Tag__639217692601576181";
       "IO_Buffer_DB".DI[301] := "Tag__639217692601764420";
       "IO_Buffer_DB".DI[302] := "Tag__639217692601904130";
       "IO_Buffer_DB".DI[303] := "Tag__639217692601921632";
       "IO_Buffer_DB".DI[304] := "Tag__639217692602082038";
       "IO_Buffer_DB".DI[305] := "Tag__639217692602243355";
       "IO_Buffer_DB".DI[306] := "Tag__639217692602403696";
       "IO_Buffer_DB".DI[307] := "Tag__639217692602403697";
       "IO_Buffer_DB".DI[308] := "Tag__639217692602561458";
       "IO_Buffer_DB".DI[309] := "Tag__639217692602720965";
       "IO_Buffer_DB".DI[310] := "Tag__639217692602881697";
       "IO_Buffer_DB".DI[311] := "Tag__639217692602881698";
       "IO_Buffer_DB".DI[312] := "Tag__639217692603041227";
       "IO_Buffer_DB".DI[313] := "Tag__639217692603201062";
       "IO_Buffer_DB".DI[314] := "Tag__639217692603432857";
       "IO_Buffer_DB".DI[315] := "Tag__639217692603526128";
       "IO_Buffer_DB".DI[316] := "Tag__639217692603677627";
       "IO_Buffer_DB".DI[317] := "Tag__639217692603839177";
       "IO_Buffer_DB".DI[318] := "Tag__639217692603998759";
       "IO_Buffer_DB".DI[319] := "Tag__639217692603998760";
       "IO_Buffer_DB".DI[320] := "Tag__639217692604301271";
       "IO_Buffer_DB".DI[321] := "Tag__639217692604446823";
       "IO_Buffer_DB".DI[322] := "Tag__639217692604524554";
       "IO_Buffer_DB".DI[323] := "Tag__639217692604674613";
       "IO_Buffer_DB".DI[324] := "Tag__639217692604834416";
       "IO_Buffer_DB".DI[325] := "Tag__639217692605944492";
       "IO_Buffer_DB".DI[326] := "Tag__639217692606105425";
       "IO_Buffer_DB".DI[327] := "Tag__639217692606105426";
       "IO_Buffer_DB".DI[328] := "Tag__639217692606285541";
       "IO_Buffer_DB".DI[329] := "Tag__639217692606426194";
       "IO_Buffer_DB".DI[330] := "Tag__639217692606584564";
       "IO_Buffer_DB".DI[331] := "Tag__639217692606742338";
       "IO_Buffer_DB".DI[332] := "Tag__639217692606904136";
       "IO_Buffer_DB".DI[333] := "Tag__639217692607062435";
       "IO_Buffer_DB".DI[334] := "Tag__639217692607224125";
       "IO_Buffer_DB".DI[335] := "Tag__639217692607224126";
       "IO_Buffer_DB".DI[336] := "Tag__639217692607485341";
       "IO_Buffer_DB".DI[337] := "Tag__639217692607543000";
       "IO_Buffer_DB".DI[338] := "Tag__639217692607763945";
       "IO_Buffer_DB".DI[339] := "Tag__639217692607861770";
       "IO_Buffer_DB".DI[340] := "Tag__639217692608018680";
       "IO_Buffer_DB".DI[341] := "Tag__639217692608018681";
       "IO_Buffer_DB".DI[342] := "Tag__639217692608238678";
       "IO_Buffer_DB".DI[343] := "Tag__639217692608335365";
       "IO_Buffer_DB".DI[344] := "Tag__639217692608493637";
       "IO_Buffer_DB".DI[345] := "Tag__639217692608653174";
       "IO_Buffer_DB".DI[346] := "Tag__639217692608812275";
       "IO_Buffer_DB".DI[347] := "Tag__639217692608812276";
       "IO_Buffer_DB".DI[348] := "Tag__639217692609128733";
       "IO_Buffer_DB".DI[349] := "Tag__639217692609128734";
       "IO_Buffer_DB".DI[350] := "Tag__639217692609289890";
       "IO_Buffer_DB".DI[351] := "Tag__639217692609532283";
       "IO_Buffer_DB".DI[352] := "Tag__639217692609702548";
       "IO_Buffer_DB".DI[353] := "Tag__639217692609862538";
       "IO_Buffer_DB".DI[354] := "Tag__639217692609862539";
       "IO_Buffer_DB".DI[355] := "Tag__639217692610182631";
       "IO_Buffer_DB".DI[356] := "Tag__639217692610182632";
       "IO_Buffer_DB".DI[357] := "Tag__639217692610403611";
       "IO_Buffer_DB".DI[358] := "Tag__639217692610501805";
       "IO_Buffer_DB".DI[359] := "Tag__639217692610661275";
       "IO_Buffer_DB".DI[360] := "Tag__639217692610661276";
       "IO_Buffer_DB".DI[361] := "Tag__639217692610983046";
       "IO_Buffer_DB".DI[362] := "Tag__639217692610983047";
       "IO_Buffer_DB".DI[363] := "Tag__639217692611192346";
       "IO_Buffer_DB".DI[364] := "Tag__639217692611310653";
       "IO_Buffer_DB".DI[365] := "Tag__639217692611461334";
       "IO_Buffer_DB".DI[366] := "Tag__639217692611622448";
       "IO_Buffer_DB".DI[367] := "Tag__639217692611781748";
       "IO_Buffer_DB".DI[368] := "Tag__639217692611781749";

       // === DIGITAL OUTPUTS: IO_Buffer_DB.DQ[1..208] -> real %Q bits ===
       // -- AFT DQ modules --
       "Tag__639217692612263475" := "IO_Buffer_DB".DQ[1];
       "Tag__639217692612423650" := "IO_Buffer_DB".DQ[2];
       "Tag__639217692612585355" := "IO_Buffer_DB".DQ[3];
       "Tag__639217692612746418" := "IO_Buffer_DB".DQ[4];
       "Tag__639217692612905975" := "IO_Buffer_DB".DQ[5];
       "Tag__639217692612905976" := "IO_Buffer_DB".DQ[6];
       "Tag__639217692613224334" := "IO_Buffer_DB".DQ[7];
       "Tag__639217692613431048" := "IO_Buffer_DB".DQ[8];
       "Tag__639217692613549459" := "IO_Buffer_DB".DQ[9];
       "Tag__639217692613549460" := "IO_Buffer_DB".DQ[10];
       "Tag__639217692613700358" := "IO_Buffer_DB".DQ[11];
       "Tag__639217692613860481" := "IO_Buffer_DB".DQ[12];
       "Tag__639217692614018559" := "IO_Buffer_DB".DQ[13];
       "Tag__639217692614298000" := "IO_Buffer_DB".DQ[14];
       "Tag__639217692614480374" := "IO_Buffer_DB".DQ[15];
       "Tag__639217692614684823" := "IO_Buffer_DB".DQ[16];
       "Tag__639217692614993876" := "IO_Buffer_DB".DQ[17];
       "Tag__639217692615192661" := "IO_Buffer_DB".DQ[18];
       "Tag__639217692615372374" := "IO_Buffer_DB".DQ[19];
       "Tag__639217692615821386" := "IO_Buffer_DB".DQ[20];
       "Tag__639217692615982422" := "IO_Buffer_DB".DQ[21];
       "Tag__639217692616141851" := "IO_Buffer_DB".DQ[22];
       "Tag__639217692616362637" := "IO_Buffer_DB".DQ[23];
       "Tag__639217692616460481" := "IO_Buffer_DB".DQ[24];
       "Tag__639217692616782087" := "IO_Buffer_DB".DQ[25];
       "Tag__639217692616782088" := "IO_Buffer_DB".DQ[26];
       "Tag__639217692616940617" := "IO_Buffer_DB".DQ[27];
       "Tag__639217692617097153" := "IO_Buffer_DB".DQ[28];
       "Tag__639217692617257965" := "IO_Buffer_DB".DQ[29];
       "Tag__639217692617425635" := "IO_Buffer_DB".DQ[30];
       "Tag__639217692617581306" := "IO_Buffer_DB".DQ[31];
       "Tag__639217692617739154" := "IO_Buffer_DB".DQ[32];
       "Tag__639217692617899719" := "IO_Buffer_DB".DQ[33];
       "Tag__639217692618058569" := "IO_Buffer_DB".DQ[34];
       "Tag__639217692618215933" := "IO_Buffer_DB".DQ[35];
       "Tag__639217692618373391" := "IO_Buffer_DB".DQ[36];
       "Tag__639217692618554770" := "IO_Buffer_DB".DQ[37];
       "Tag__639217692618760680" := "IO_Buffer_DB".DQ[38];
       "Tag__639217692618931105" := "IO_Buffer_DB".DQ[39];
       "Tag__639217692619091004" := "IO_Buffer_DB".DQ[40];
       "Tag__639217692619165425" := "IO_Buffer_DB".DQ[41];
       "Tag__639217692619325369" := "IO_Buffer_DB".DQ[42];
       "Tag__639217692619487118" := "IO_Buffer_DB".DQ[43];
       "Tag__639217692619487119" := "IO_Buffer_DB".DQ[44];
       "Tag__639217692619648292" := "IO_Buffer_DB".DQ[45];
       "Tag__639217692619808948" := "IO_Buffer_DB".DQ[46];
       "Tag__639217692620036810" := "IO_Buffer_DB".DQ[47];
       "Tag__639217692620197299" := "IO_Buffer_DB".DQ[48];
       "Tag__639217692620337293" := "IO_Buffer_DB".DQ[49];
       "Tag__639217692620357294" := "IO_Buffer_DB".DQ[50];
       "Tag__639217692620515379" := "IO_Buffer_DB".DQ[51];
       "Tag__639217692620675332" := "IO_Buffer_DB".DQ[52];
       "Tag__639217692620835634" := "IO_Buffer_DB".DQ[53];
       "Tag__639217692620992973" := "IO_Buffer_DB".DQ[54];
       "Tag__639217692621152065" := "IO_Buffer_DB".DQ[55];
       "Tag__639217692621309565" := "IO_Buffer_DB".DQ[56];
       "Tag__639217692621469714" := "IO_Buffer_DB".DQ[57];
       "Tag__639217692621469715" := "IO_Buffer_DB".DQ[58];
       "Tag__639217692621630499" := "IO_Buffer_DB".DQ[59];
       "Tag__639217692621906549" := "IO_Buffer_DB".DQ[60];
       "Tag__639217692621950360" := "IO_Buffer_DB".DQ[61];
       "Tag__639217692622111179" := "IO_Buffer_DB".DQ[62];
       "Tag__639217692622292619" := "IO_Buffer_DB".DQ[63];
       "Tag__639217692622426875" := "IO_Buffer_DB".DQ[64];
       // -- MID DQ modules --
       "Tag__639217692622426876" := "IO_Buffer_DB".DQ[65];
       "Tag__639217692622587394" := "IO_Buffer_DB".DQ[66];
       "Tag__639217692622746975" := "IO_Buffer_DB".DQ[67];
       "Tag__639217692622906735" := "IO_Buffer_DB".DQ[68];
       "Tag__639217692623064209" := "IO_Buffer_DB".DQ[69];
       "Tag__639217692623222595" := "IO_Buffer_DB".DQ[70];
       "Tag__639217692623222596" := "IO_Buffer_DB".DQ[71];
       "Tag__639217692623428677" := "IO_Buffer_DB".DQ[72];
       "Tag__639217692623552568" := "IO_Buffer_DB".DQ[73];
       "Tag__639217692623706024" := "IO_Buffer_DB".DQ[74];
       "Tag__639217692623866625" := "IO_Buffer_DB".DQ[75];
       "Tag__639217692624026402" := "IO_Buffer_DB".DQ[76];
       "Tag__639217692624188100" := "IO_Buffer_DB".DQ[77];
       "Tag__639217692624296413" := "IO_Buffer_DB".DQ[78];
       "Tag__639217692624349590" := "IO_Buffer_DB".DQ[79];
       "Tag__639217692624607979" := "IO_Buffer_DB".DQ[80];
       "Tag__639217692624665644" := "IO_Buffer_DB".DQ[81];
       "Tag__639217692624979691" := "IO_Buffer_DB".DQ[82];
       "Tag__639217692625112094" := "IO_Buffer_DB".DQ[83];
       "Tag__639217692625921588" := "IO_Buffer_DB".DQ[84];
       "Tag__639217692626087431" := "IO_Buffer_DB".DQ[85];
       "Tag__639217692626253351" := "IO_Buffer_DB".DQ[86];
       "Tag__639217692626352897" := "IO_Buffer_DB".DQ[87];
       "Tag__639217692626510009" := "IO_Buffer_DB".DQ[88];
       "Tag__639217692626671657" := "IO_Buffer_DB".DQ[89];
       "Tag__639217692626671658" := "IO_Buffer_DB".DQ[90];
       "Tag__639217692626833520" := "IO_Buffer_DB".DQ[91];
       "Tag__639217692626994806" := "IO_Buffer_DB".DQ[92];
       "Tag__639217692627254988" := "IO_Buffer_DB".DQ[93];
       "Tag__639217692627312671" := "IO_Buffer_DB".DQ[94];
       "Tag__639217692627473354" := "IO_Buffer_DB".DQ[95];
       "Tag__639217692627673115" := "IO_Buffer_DB".DQ[96];
       "Tag__639217692627811109" := "IO_Buffer_DB".DQ[97];
       "Tag__639217692627949093" := "IO_Buffer_DB".DQ[98];
       "Tag__639217692628089666" := "IO_Buffer_DB".DQ[99];
       "Tag__639217692628107166" := "IO_Buffer_DB".DQ[100];
       "Tag__639217692628336120" := "IO_Buffer_DB".DQ[101];
       "Tag__639217692628492917" := "IO_Buffer_DB".DQ[102];
       "Tag__639217692628623290" := "IO_Buffer_DB".DQ[103];
       "Tag__639217692628761042" := "IO_Buffer_DB".DQ[104];
       "Tag__639217692628899816" := "IO_Buffer_DB".DQ[105];
       "Tag__639217692628972569" := "IO_Buffer_DB".DQ[106];
       "Tag__639217692629072663" := "IO_Buffer_DB".DQ[107];
       "Tag__639217692629316047" := "IO_Buffer_DB".DQ[108];
       "Tag__639217692629373725" := "IO_Buffer_DB".DQ[109];
       "Tag__639217692629533777" := "IO_Buffer_DB".DQ[110];
       "Tag__639217692629693574" := "IO_Buffer_DB".DQ[111];
       "Tag__639217692629851555" := "IO_Buffer_DB".DQ[112];
       "Tag__639217692630008442" := "IO_Buffer_DB".DQ[113];
       "Tag__639217692630168713" := "IO_Buffer_DB".DQ[114];
       "Tag__639217692630329520" := "IO_Buffer_DB".DQ[115];
       "Tag__639217692630490637" := "IO_Buffer_DB".DQ[116];
       "Tag__639217692630661059" := "IO_Buffer_DB".DQ[117];
       "Tag__639217692630807879" := "IO_Buffer_DB".DQ[118];
       "Tag__639217692630939597" := "IO_Buffer_DB".DQ[119];
       "Tag__639217692631073684" := "IO_Buffer_DB".DQ[120];
       "Tag__639217692631183654" := "IO_Buffer_DB".DQ[121];
       "Tag__639217692631183655" := "IO_Buffer_DB".DQ[122];
       "Tag__639217692631342517" := "IO_Buffer_DB".DQ[123];
       "Tag__639217692631504108" := "IO_Buffer_DB".DQ[124];
       "Tag__639217692631664286" := "IO_Buffer_DB".DQ[125];
       "Tag__639217692631824426" := "IO_Buffer_DB".DQ[126];
       "Tag__639217692631981364" := "IO_Buffer_DB".DQ[127];
       "Tag__639217692631981365" := "IO_Buffer_DB".DQ[128];
       // -- FWD DQ modules --
       "Tag__639217692632142556" := "IO_Buffer_DB".DQ[129];
       "Tag__639217692632301255" := "IO_Buffer_DB".DQ[130];
       "Tag__639217692632461403" := "IO_Buffer_DB".DQ[131];
       "Tag__639217692632622376" := "IO_Buffer_DB".DQ[132];
       "Tag__639217692632622377" := "IO_Buffer_DB".DQ[133];
       "Tag__639217692632781836" := "IO_Buffer_DB".DQ[134];
       "Tag__639217692633119556" := "IO_Buffer_DB".DQ[135];
       "Tag__639217692633257667" := "IO_Buffer_DB".DQ[136];
       "Tag__639217692633257668" := "IO_Buffer_DB".DQ[137];
       "Tag__639217692633606974" := "IO_Buffer_DB".DQ[138];
       "Tag__639217692633797544" := "IO_Buffer_DB".DQ[139];
       "Tag__639217692633935297" := "IO_Buffer_DB".DQ[140];
       "Tag__639217692634052982" := "IO_Buffer_DB".DQ[141];
       "Tag__639217692634250953" := "IO_Buffer_DB".DQ[142];
       "Tag__639217692634367505" := "IO_Buffer_DB".DQ[143];
       "Tag__639217692634526933" := "IO_Buffer_DB".DQ[144];
       "Tag__639217692634686575" := "IO_Buffer_DB".DQ[145];
       "Tag__639217692634847392" := "IO_Buffer_DB".DQ[146];
       "Tag__639217692635084699" := "IO_Buffer_DB".DQ[147];
       "Tag__639217692635166263" := "IO_Buffer_DB".DQ[148];
       "Tag__639217692635324026" := "IO_Buffer_DB".DQ[149];
       "Tag__639217692635482506" := "IO_Buffer_DB".DQ[150];
       "Tag__639217692635482507" := "IO_Buffer_DB".DQ[151];
       "Tag__639217692635642498" := "IO_Buffer_DB".DQ[152];
       "Tag__639217692635802017" := "IO_Buffer_DB".DQ[153];
       "Tag__639217692636027800" := "IO_Buffer_DB".DQ[154];
       "Tag__639217692636167857" := "IO_Buffer_DB".DQ[155];
       "Tag__639217692636298889" := "IO_Buffer_DB".DQ[156];
       "Tag__639217692636348888" := "IO_Buffer_DB".DQ[157];
       "Tag__639217692636549597" := "IO_Buffer_DB".DQ[158];
       "Tag__639217692636666551" := "IO_Buffer_DB".DQ[159];
       "Tag__639217692636827995" := "IO_Buffer_DB".DQ[160];
       "Tag__639217692636988786" := "IO_Buffer_DB".DQ[161];
       "Tag__639217692636988787" := "IO_Buffer_DB".DQ[162];
       "Tag__639217692637150621" := "IO_Buffer_DB".DQ[163];
       "Tag__639217692637311136" := "IO_Buffer_DB".DQ[164];
       "Tag__639217692637471435" := "IO_Buffer_DB".DQ[165];
       "Tag__639217692637631790" := "IO_Buffer_DB".DQ[166];
       "Tag__639217692637789494" := "IO_Buffer_DB".DQ[167];
       "Tag__639217692637950184" := "IO_Buffer_DB".DQ[168];
       "Tag__639217692637950185" := "IO_Buffer_DB".DQ[169];
       "Tag__639217692638109462" := "IO_Buffer_DB".DQ[170];
       "Tag__639217692638276714" := "IO_Buffer_DB".DQ[171];
       "Tag__639217692638427229" := "IO_Buffer_DB".DQ[172];
       "Tag__639217692638586533" := "IO_Buffer_DB".DQ[173];
       "Tag__639217692638747466" := "IO_Buffer_DB".DQ[174];
       "Tag__639217692638904386" := "IO_Buffer_DB".DQ[175];
       "Tag__639217692639063833" := "IO_Buffer_DB".DQ[176];
       "Tag__639217692639078981" := "IO_Buffer_DB".DQ[177];
       "Tag__639217692639243768" := "IO_Buffer_DB".DQ[178];
       "Tag__639217692639383298" := "IO_Buffer_DB".DQ[179];
       "Tag__639217692639542163" := "IO_Buffer_DB".DQ[180];
       "Tag__639217692639701541" := "IO_Buffer_DB".DQ[181];
       "Tag__639217692639892825" := "IO_Buffer_DB".DQ[182];
       "Tag__639217692640016631" := "IO_Buffer_DB".DQ[183];
       "Tag__639217692640016632" := "IO_Buffer_DB".DQ[184];
       "Tag__639217692640175734" := "IO_Buffer_DB".DQ[185];
       "Tag__639217692640332797" := "IO_Buffer_DB".DQ[186];
       "Tag__639217692640492541" := "IO_Buffer_DB".DQ[187];
       "Tag__639217692640652754" := "IO_Buffer_DB".DQ[188];
       "Tag__639217692640652755" := "IO_Buffer_DB".DQ[189];
       "Tag__639217692640812694" := "IO_Buffer_DB".DQ[190];
       "Tag__639217692640972759" := "IO_Buffer_DB".DQ[191];
       "Tag__639217692641133541" := "IO_Buffer_DB".DQ[192];
       "Tag__639217692641370581" := "IO_Buffer_DB".DQ[193];
       "Tag__639217692641539941" := "IO_Buffer_DB".DQ[194];
       "Tag__639217692641669868" := "IO_Buffer_DB".DQ[195];
       "Tag__639217692641679864" := "IO_Buffer_DB".DQ[196];
       "Tag__639217692641838308" := "IO_Buffer_DB".DQ[197];
       "Tag__639217692641998720" := "IO_Buffer_DB".DQ[198];
       "Tag__639217692642156578" := "IO_Buffer_DB".DQ[199];
       "Tag__639217692642313321" := "IO_Buffer_DB".DQ[200];
       "Tag__639217692642472571" := "IO_Buffer_DB".DQ[201];
       "Tag__639217692642631876" := "IO_Buffer_DB".DQ[202];
       "Tag__639217692642631877" := "IO_Buffer_DB".DQ[203];
       "Tag__639217692642792640" := "IO_Buffer_DB".DQ[204];
       "Tag__639217692642950472" := "IO_Buffer_DB".DQ[205];
       "Tag__639217692643191744" := "IO_Buffer_DB".DQ[206];
       "Tag__639217692643266837" := "IO_Buffer_DB".DQ[207];
       "Tag__639217692643431479" := "IO_Buffer_DB".DQ[208];
END_FUNCTION

FUNCTION "FC_IoMapper" : Void   // FC1, SCL
{ S7_Optimized_Access := 'TRUE' }
VERSION : 0.1
// NOT YET WIRED INTO Main[OB1] - built and compiles clean, but deliberately not called anywhere yet. Two things need to happen first: (1) confirm real physical %I/%Q addresses for the ET200SP DI/DQ modules - an address probe run 2026-08-08 found every DI/DQ module reporting StartAddress=-1, meaning either they are not actually seated in real rack slots or addresses simply are not assigned until a real download; needs visual confirmation in TIA's Device view before anything here can read real hardware. (2) FB_ValveLoop's own simulated OpenFB/ClosedFB writes (Section 1 "Motion Simulation") need a guard added so they skip any valve that has a real channel assigned here, otherwise the simulation will keep overwriting whatever this mapper writes. Until both are done, every valve stays on symbolic simulation exactly as today - this block is inert scaffolding, safe to have present without affecting the running demo.
// stored: AutoNumber true, IsIECCheckEnabled false, SetENOAutomatically false, UDAEnableTagReadback false
   VAR_TEMP
      i : Int;
      stationDown : Bool;
   END_VAR
BEGIN
// Network 1

       // Dynamic I/O Mapper: translates each valve's abstract channel-index config
       // (Valve_Channels_DB's six flat OpenFbChannel[]/ClosedFbChannel[]/etc arrays) into real feedback/health bits by looking them up in
       // IO_Buffer_DB.DI[], and writes commanded outputs into IO_Buffer_DB.DQ[] the same way.
       // A channel value of 0 means "not assigned" - that field is simply left untouched, so an
       // unconfigured channel never overwrites a valve's simulated status with a false FALSE.
       FOR #i := 1 TO 89 DO
           // Which station carries this valve. Confirmed against Valve_Channels_DB rather than
           // assumed: valves 1-27 use DI channels 1-108 (AFT provides 1-112), 28-54 use 113-220
           // (MID provides 113-224), 55-89 use 225-364 (FWD provides 225-368).
           #stationDown := (#i <= 27 AND "Diag_DB".AftLost)
                        OR (#i > 27 AND #i <= 54 AND "Diag_DB".MidLost)
                        OR (#i > 54 AND "Diag_DB".FwdLost);

           // NOT #stationDown is the important half of this guard. When a station is off the network
           // its input data is not a report from the field, and what the process image holds instead
           // is not something this project has been able to establish - Siemens' own documentation
           // was not found to say whether inputs go to zero or freeze at their last value, and it
           // cannot be tested in simulation because PLCSIM runs no PROFINET. Both possibilities are
           // bad in different ways: zeros make every valve on the station report no position and not
           // healthy, which is ~54 alarms burying the one that explains them; frozen values make a
           // dead station look perfectly normal.
           //
           // Skipping the copy removes the question. Valve[i].OpenFB/ClosedFB/Healthy/LocalMode
           // simply keep the values they last had, which is the last real report from the field -
           // the thing an operator actually needs when a station drops, since knowing whether a
           // ballast line was open or shut is the first question asked. And because Healthy stays
           // TRUE and the position stays valid, the Unhealthy and Loss-of-Position alarms do not
           // fire for the whole station, leaving the RIO station alarm standing on its own.
           //
           // Travel timeouts are deliberately NOT suppressed. If someone commands a valve on a dead
           // station, nothing moves and FailOpen/FailClose is the correct thing to say - that is one
           // alarm about one deliberate action, not a flood.
           IF "Valves_DB".Valve[#i].Configured AND NOT #stationDown THEN
               IF "Valve_Channels_DB".OpenFbChannel[#i] > 0 THEN
                   "Valves_DB".Valve[#i].OpenFB := "IO_Buffer_DB".DI["Valve_Channels_DB".OpenFbChannel[#i]];
               END_IF;
               IF "Valve_Channels_DB".ClosedFbChannel[#i] > 0 THEN
                   "Valves_DB".Valve[#i].ClosedFB := "IO_Buffer_DB".DI["Valve_Channels_DB".ClosedFbChannel[#i]];
               END_IF;
               IF "Valve_Channels_DB".HealthyChannel[#i] > 0 THEN
                   "Valves_DB".Valve[#i].Healthy := "IO_Buffer_DB".DI["Valve_Channels_DB".HealthyChannel[#i]];
               END_IF;
               // Double-indication safety trip, re-applied here on purpose: FB_ValveLoop already
               // checks this earlier in the same scan, but for a real-channel valve this Healthy
               // write above runs AFTER that check and would silently undo it - a real valve with
               // both limit switches made (physically impossible, a wiring/sensor fault) would show
               // Healthy=TRUE if the real Healthy channel itself doesn't happen to also be false.
               // Found by reasoning through the watch-table test 2026-08-14, not observed live (that
               // test only forced OpenFB, never both at once) - fixing before it's ever hit for real.
               IF "Valves_DB".Valve[#i].OpenFB AND "Valves_DB".Valve[#i].ClosedFB THEN
                   "Valves_DB".Valve[#i].Healthy := FALSE;
               END_IF;
               IF "Valve_Channels_DB".LocalModeChannel[#i] > 0 THEN
                   "Valves_DB".Valve[#i].LocalMode := "IO_Buffer_DB".DI["Valve_Channels_DB".LocalModeChannel[#i]];
               END_IF;
           END_IF;
           // Outputs are driven UNCONDITIONALLY - deliberately outside the Configured guard above.
           // That guard exists to protect a simulated valve's feedbacks from being overwritten by a
           // real DI; it has no business gating the outputs. When it did, de-configuring a valve
           // mid-travel froze its DQ bit at whatever it was last written to, and FC_PhysicalIoCopy
           // kept copying that stale TRUE to the real %Q forever - a relay energised with nothing
           // managing it. FB_ValveLoop now forces OpenValve/CloseValve FALSE for any unconfigured
           // valve, so writing DQ every scan regardless is what actually de-energises the output.
           IF "Valve_Channels_DB".OpenCmdChannel[#i] > 0 THEN
               "IO_Buffer_DB".DQ["Valve_Channels_DB".OpenCmdChannel[#i]] := "Valves_DB".Valve[#i].OpenValve;
           END_IF;
           IF "Valve_Channels_DB".CloseCmdChannel[#i] > 0 THEN
               "IO_Buffer_DB".DQ["Valve_Channels_DB".CloseCmdChannel[#i]] := "Valves_DB".Valve[#i].CloseValve;
           END_IF;
       END_FOR;
END_FUNCTION

ORGANIZATION_BLOCK "RackOrStationFailure"   // OB86, SCL, RackOrStationFailure
{ S7_Optimized_Access := 'TRUE' }
VERSION : 0.1
// stored: IsIECCheckEnabled false, SetENOAutomatically false
   VAR_INPUT
      LADDR : HW_DEVICE;   // Hardware identifier
      Event_Class : Byte;   // Event class
      Fault_ID : Byte;   // Fault identifier
   END_VAR
BEGIN
END_ORGANIZATION_BLOCK

ORGANIZATION_BLOCK "DiagnosticErrorInterrupt"   // OB82, SCL, DiagnosticErrorInterrupt
{ S7_Optimized_Access := 'TRUE' }
VERSION : 0.1
// Called by the CPU when an I/O module reports a diagnostic. Latches Diag_DB.ModuleFault, which FB_ValveLoop turns into HwHealthy[5] and thence HwWord bit 4, driving the existing System_IO_Module_Fault alarm. Deliberately does not decode IO_State - see the body comment.
// stored: IsIECCheckEnabled false, SetENOAutomatically false
   VAR_INPUT
      IO_State : Word;   // IO state of the HW object
      LADDR : HW_ANY;   // Hardware identifier
      Channel : UInt;   // Channel number
      MultiError : Bool;   // =true if more than one error is present
   END_VAR
   VAR_TEMP
      id : UInt;
   END_VAR
BEGIN

   // Called by the CPU when an I/O module raises a diagnostic: its 24 V supply
   // failing, a DQ output short-circuited to L+ or to ground, a parameter error, or
   // a wire break where that is ever enabled. Those diagnostics were switched on
   // across all 36 modules on 2026-09-06 - they ship DISABLED, which is why nothing
   // would have reached this block even if it had existed earlier.
   //
   // WHY THIS BLOCK DOES NOT DECODE #IO_State
   //
   // The same OB fires when a fault APPEARS and again when it GOES AWAY, and
   // #IO_State is what separates the two. Its bit meanings could not be confirmed
   // from any reachable Siemens source, and this block cannot be tested here:
   // PLCSIM does not simulate module-level diagnostics, for the same reason it does
   // not simulate the station events OB86 handles (handoff item 11).
   //
   // Guessing the polarity would risk precisely the failure OB86's own comment
   // warns about - clearing the flag on failure and setting it on recovery, giving
   // a system that reports healthy exactly when it is not. So this block does not
   // guess. ModuleFault LATCHES on any event and clears only via ModuleFaultAck.
   //
   // The worst case is a stale fault sitting after a module has recovered: visible,
   // irritating, and safe. The opposite error is silent. UnexpMove and DirFault
   // already latch for the same reason.
   //
   // Everything is stored RAW and undecoded so the bit meanings can be LEARNED from
   // the real panel rather than guessed now: pull a module and read
   // LastModuleIoState, plug it back in and read it again. Two observations settle
   // what the documentation would not.

   "Diag_DB".ModuleFault := TRUE;

   #id := #LADDR;
   "Diag_DB".LastModuleLaddr := #id;
   "Diag_DB".LastModuleIoState := #IO_State;
   "Diag_DB".LastModuleChannel := #Channel;
   "Diag_DB".LastModuleMultiError := #MultiError;

   // Saturating, not wrapping. An Int rolling past 32767 into negative would read as
   // a different kind of fault to whoever is looking at it, and the exact count that
   // far out says nothing the latched flag has not already said. What the count is
   // genuinely for is spotting a module that is CHATTERING - rising steadily while
   // ModuleFault has never been cleared.
   IF "Diag_DB".ModuleEventCount < 32767 THEN
       "Diag_DB".ModuleEventCount := "Diag_DB".ModuleEventCount + 1;
   END_IF;
END_ORGANIZATION_BLOCK

FUNCTION_BLOCK "FB_ValveLogic"   // FB3, SCL
{ S7_Optimized_Access := 'TRUE' }
VERSION : 0.1
// stored: AutoNumber true, IsIECCheckEnabled false, IsRetainMemResEnabled false, MemoryReserve 100, SetENOAutomatically false, UDAEnableTagReadback false
   VAR_IN_OUT
      Valve : "Valve_IO";
   END_VAR
BEGIN
   IF #Valve.Configured THEN

       // Mutual exclusion — Close takes priority if both are somehow TRUE
       IF #Valve.CloseCmd THEN
           #Valve.OpenCmd := FALSE;
       END_IF;
       IF #Valve.OpenCmd THEN
           #Valve.CloseCmd := FALSE;
       END_IF;

       // OPEN side
       IF #Valve.OpenCmd AND NOT #Valve.LocalMode AND #Valve.Healthy THEN
           #Valve.OpenValve := TRUE;
       ELSE
           #Valve.OpenValve := FALSE;
       END_IF;

       #Valve.TimerOpen(IN := #Valve.OpenValve,
                        PT := T#5s);
       IF #Valve.TimerOpen.Q THEN
           #Valve.OpenFB := TRUE;
           #Valve.ClosedFB := FALSE;
       END_IF;

       // CLOSE side
       IF #Valve.CloseCmd AND NOT #Valve.LocalMode AND #Valve.Healthy THEN
           #Valve.CloseValve := TRUE;
       ELSE
           #Valve.CloseValve := FALSE;
       END_IF;

       #Valve.TimerClose(IN := #Valve.CloseValve,
                         PT := T#5s);
       IF #Valve.TimerClose.Q THEN
           #Valve.ClosedFB := TRUE;
           #Valve.OpenFB := FALSE;
       END_IF;

   ELSE
       // Not configured — force everything safe/off
       #Valve.OpenValve := FALSE;
       #Valve.CloseValve := FALSE;
   END_IF;
END_FUNCTION_BLOCK

FUNCTION_BLOCK "FB_HMI_MIirror"   // FB5, SCL
{ S7_Optimized_Access := 'TRUE' }
VERSION : 0.1
// stored: AutoNumber true, IsIECCheckEnabled false, IsRetainMemResEnabled false, MemoryReserve 100, SetENOAutomatically false, UDAEnableTagReadback false
   VAR
      Lastindex : Int;
   END_VAR
   VAR_TEMP
      idx : Int;
   END_VAR
BEGIN
   // Read selected index and clamp to valid range (1..88)
   #idx := "HMI_Interface_DB".SelectedValveIndex;

   IF #idx < 1 THEN
       #idx := 1;
   ELSIF #idx > 88 THEN
       #idx := 88;
   END_IF;

   // Detect index change -> reset stale commands before mirroring
   IF #idx <> #Lastindex THEN
       "HMI_Interface_DB".OpenCmd := FALSE;
       "HMI_Interface_DB".CloseCmd := FALSE;
       #Lastindex := #idx;
   END_IF;

   // Mirror PLC -> HMI (feedback)
   "HMI_Interface_DB".OpenFB := "Valves_DB".Valve[#idx].OpenFB;
   "HMI_Interface_DB".ClosedFB := "Valves_DB".Valve[#idx].ClosedFB;
   "HMI_Interface_DB".Healthy := "Valves_DB".Valve[#idx].Healthy;
   "HMI_Interface_DB".LocalMode := "Valves_DB".Valve[#idx].LocalMode;

   // Mirror HMI -> PLC (commands)
   "Valves_DB".Valve[#idx].OpenCmd := "HMI_Interface_DB".OpenCmd;
   "Valves_DB".Valve[#idx].CloseCmd := "HMI_Interface_DB".CloseCmd;
END_FUNCTION_BLOCK

FUNCTION_BLOCK "FB_ValveControl"   // FB1, LAD
{ S7_Optimized_Access := 'TRUE' }
VERSION : 0.1
// stored: AutoNumber true, IsIECCheckEnabled false, IsRetainMemResEnabled false, MemoryReserve 100, SetENOAutomatically false, UDAEnableTagReadback false
   VAR_INPUT
      OpenCmd : Bool;
      CloseCmd : Bool;
      LocalMode : Bool;
      Healthy : Bool;
      OpenFB : Bool;
      ClosedFB : Bool;
   END_VAR
   VAR_OUTPUT
      OpenValve : Bool;
      CloseValve : Bool;
   END_VAR
BEGIN

REGION Network 1
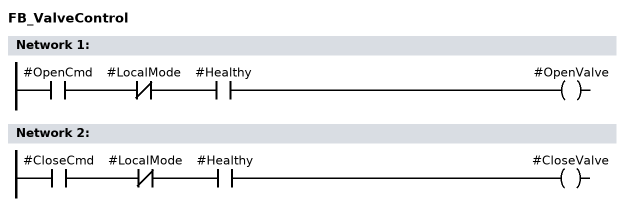
   RUNG wire#powerrail
      Contact( #OpenCmd )
      I_Contact( #LocalMode )
      Contact( #Healthy )
      Coil( #OpenValve )
   END_RUNG
   // the same network as SCL:
   #OpenValve := #OpenCmd AND NOT #LocalMode AND #Healthy;
END_REGION

REGION Network 2
   RUNG wire#powerrail
      Contact( #CloseCmd )
      I_Contact( #LocalMode )
      Contact( #Healthy )
      Coil( #CloseValve )
   END_RUNG
   // the same network as SCL:
   #CloseValve := #CloseCmd AND NOT #LocalMode AND #Healthy;
END_REGION
END_FUNCTION_BLOCK
